TYPE ST_RT6D :
STRUCT
	x : REAL;
	y : REAL;
	z : REAL;
	rotMatrix : ARRAY [0..8] OF REAL;
END_STRUCT
END_TYPE

(* stored: Version 1.1.0.1, ProductVersion 3.1.4026.8
   DUT ST_RT6D: Id {3167e8f5-29b6-4182-8974-6a201a5fdfda} *)
